PROGRAM _1000_PRG_Homing
VAR_IN_OUT
    CurrentStep : ActiveStep;  // Shared step structure with state machine
	NextStep: DINT; // Next step to be modified by sequences
END_VAR

VAR_INPUT
    StepTimerSeconds : DINT;   // Timer value from state machine
    RetrySignal : BOOL;        // Retry signal from state machine
    StateMachineStatus : ST_SM_Status;  // Complete state machine status
END_VAR


VAR
    // Step function blocks for homing sequence
    fbStep1000 : FB_SequenceStep;  // Home Initialize
    fbStep1002 : FB_SequenceStep;  // Home Execute
    
    // Step permissives (simulation for testing)
    step1000Perms : INT := -1;     // All OK for step 1000
    step1002Perms : INT := -1;     // All OK for step 1002
    
END_VAR

//=============================================================================
// PRG_Homing - Handles HOMING state sequence (1000-1999)
//=============================================================================
// Step numbering: 1000, 1002 (even numbers)
// Fault steps: 1001, 1003 (odd numbers, +1 of original)
// NOTE: Initial step setting (CurrentStep.Step = 0) is handled in MAIN program


//=============================================================================
// STEP 1000 - HOME INITIALIZE
//=============================================================================
fbStep1000(
    inpStep := CurrentStep.Step,
    cfgStep := 1000,
    cfgNextStep := 1002,
    inpStepTimerSeconds := StepTimerSeconds,
    inpRetry := RetrySignal,
    inpStepPermissives := step1000Perms,
    cfgStepTimeout := 10,  // 10 second timeout
    inpFaultStep := FALSE,
    ActiveStep := CurrentStep
);

// Step 1000 Active Logic
IF fbStep1000.outStepActive THEN
    // Only simulate permissives if step is active but not advancing
    IF fbStep1000.outNextStep = fbStep1000.cfgStep THEN  // Step is waiting for permissives
        // Permissives simulation - Simulate based on timer
        IF StepTimerSeconds < 3 THEN
            step1000Perms := 16#FFFE;  // Bit 0 not OK (not ready yet)
        ELSE
            step1000Perms := -1;  // All permissives OK after 3 seconds
        END_IF;
    END_IF;
    
    // HMI configuration and actions
    CurrentStep.PermsHMI.Name := 'Home Initialize';
    CurrentStep.PermsHMI.Desc[0] := 'System Ready';
    CurrentStep.PermsHMI.Desc[1] := 'Home Position Clear';
    CurrentStep.PermsHMI.Desc[2] := 'Safety Systems OK';
    
    // Add any step-specific actions here
    // Example: Reset position counters, check home sensors, etc.
    
    // FB_SequenceStep determines next step automatically based on permissives
    NextStep := fbStep1000.outNextStep;
ELSE
    // Reset permissives when step is not active (ensures fresh start next time)
    step1000Perms := 16#FFFE;  // Reset to NOT OK when leaving step
END_IF;

//=============================================================================
// STEP 1002 - HOME EXECUTE
//=============================================================================
fbStep1002(
    inpStep := CurrentStep.Step,
    cfgStep := 1002,
    cfgNextStep := 999,  // 0 = sequence complete
    inpStepTimerSeconds := StepTimerSeconds,
    inpRetry := RetrySignal,
    inpStepPermissives := step1002Perms,
    cfgStepTimeout := 15,  // 15 second timeout
    inpFaultStep := FALSE,
    ActiveStep := CurrentStep
);

// Step 1002 Active Logic
IF fbStep1002.outStepActive THEN
    // Only simulate permissives if step is active but not advancing
    IF fbStep1002.outNextStep = fbStep1002.cfgStep THEN  // Step is waiting for permissives
        // Permissives simulation - Simulate based on timer
        IF StepTimerSeconds < 8 THEN
            step1002Perms := 16#FFFD;  // Bit 1 not OK (homing not complete)
        ELSE
            step1002Perms := -1;  // All permissives OK after 8 seconds
        END_IF;
    END_IF;
    
    // HMI configuration and actions
    CurrentStep.PermsHMI.Name := 'Home Execute';
    CurrentStep.PermsHMI.Desc[0] := 'Motors Enabled';
    CurrentStep.PermsHMI.Desc[1] := 'Home Sensors Active';
    CurrentStep.PermsHMI.Desc[2] := 'No Emergency Stops';
    
    // Add any step-specific actions here
    // Example: Start homing motion, monitor position feedback, etc.
    
    // FB_SequenceStep determines next step automatically based on permissives
    NextStep := fbStep1002.outNextStep;
ELSE
    // Reset permissives when step is not active (ensures fresh start next time)
    step1002Perms := 16#FFFD;  // Reset to NOT OK when leaving step
END_IF;

END_PROGRAM

(* stored: Version 1.1.0.1, ProductVersion 3.1.4024.13
   POU _1000_PRG_Homing: Id {12345678-1234-1234-1234-123456789001}, SpecialFunc None *)
